// TIA Portal V20 export
TYPE "typeNoSaftyFaultGroup"
// stored: Access Published, IsFailsafeCompliant true, Namespace Safety
   STRUCT
      noSaftyFaultGroup1 : Bool;   // Safety Device QBAD Group 1
      noSaftyFaultGroup2 : Bool;   // Safety Device QBAD Group 2
      noSaftyFaultGroup3 : Bool;   // Safety Device QBAD Group 3
   END_STRUCT;
END_TYPE
